// TIA Portal project "Lab_3" (V18)

(* hardware
DEVICE "S7-1500/ET200MP station_1"  S7-1500 station
   slot 0: "Rail_0"  Rack  6ES7 590-1***0-0AA0
   slot 1: "PLC_1"  CPU 1511-1 PN  6ES7 511-1AK00-0AB0  V1.0
      slot 3: "CPU display_1"  6ES7591-1XA00-0AA0
      slot 32768: "PROFINET interface_1"  X1
   slot 2: "CM 1542-5_1"  CM 1542-5  6GK7 542-5DX00-0XE0  V1.0
   slot 3: "DI 16x24VDC HF_1"  DI 16x24VDC HF  6ES7 521-1BH00-0AB0  V1.0
   slot 4: "DQ 16x24VDC/0.5A ST_1"  DQ 16x24VDC/0.5A ST  6ES7 522-1BH00-0AB0  V1.0
   slot 5: "AI 8xU/I/RTD/TC ST_1"  AI 8xU/I/RTD/TC ST  6ES7 531-7KF00-0AB0  V1.0
   slot 6: "AQ 4xU/I ST_1"  AQ 4xU/I ST  6ES7 532-5HD00-0AB0  V1.0
DEVICE "HMI_1"  KTP600 Basic color PN SIPLUS
   slot 0: "HMI_1"  KTP600 Basic color PN SIPLUS  6AG1 647-0AD11-2AX0  12.0.0.0
   slot 1: "HMI_RT_1"  KTP600 Basic color PN SIPLUS  6AG1 647-0AD11-2AX0  12.0.0.0
   slot 5: "HMI_1.IE_CP_1"  PROFINET Interface  12.0.0.0
      slot 1: "PROFINET Interface_1"  PROFINET Interface
         slot 1: "Port_1"  Port
*)

// ===== PLC "PLC_1"  CPU 1511-1 PN =====

VAR_GLOBAL   // PLC tag table "Default tag table"
   "Start_Pulse" AT %M0.0 : Bool;
   "En_Pulse" AT %M0.1 : Bool;
   "Low_Pulse_Active" AT %M0.2 : Bool;
   "High_Pulse_Enable" AT %M0.3 : Bool;
   "High_Pulse_Active" AT %M0.4 : Bool;
   "Low_Pulse_Enable" AT %M0.5 : Bool;
   "Pulse" AT %Q0.0 : Bool;
   "Start" AT %I0.0 : Bool;
   "Stop" AT %I0.1 : Bool;
   "Emergency" AT %I0.2 : Bool;
   "En_Bottle" AT %M2.0 : Bool;
   "R_Bottle" AT %M2.1 : Bool;
   "Finish_Bottle" AT %M2.2 : Bool;
   "Count_Bottle" AT %MW3 : Int;
   "R_Pulse" AT %M5.0 : Bool;
   "F_Pulse" AT %M5.1 : Bool;
   "Count_Pulse" AT %MW6 : Int;
   "En_PWM" AT %M8.0 : Bool;
   "Completo_PWM" AT %M8.1 : Bool;
   "T_PWM" AT %MD10 : Time;
   "E_Fill" AT %M14.0 : Bool;
   "Total_Fill" AT %M14.1 : Bool;
   "T_Fill" AT %MD15 : Time;
   "Valve" AT %M20.0 : Bool;
   "Bottles" AT %MW30 : Int;
   "Etapa" AT %M40.2 : Bool;
END_VAR

DATA_BLOCK "Generador_DB"   // DB2
{ S7_Optimized_Access := 'TRUE' }
VERSION : 0.1
// stored: InstanceOfName Generador
"Generador"
BEGIN
END_DATA_BLOCK

DATA_BLOCK "Contadores y Temporizadores_DB"   // DB3
{ S7_Optimized_Access := 'TRUE' }
VERSION : 0.1
// stored: InstanceOfName Contadores y Temporizadores
"Contadores y Temporizadores"
BEGIN
END_DATA_BLOCK

DATA_BLOCK "graph_DB"   // DB4
{ S7_Optimized_Access := 'TRUE' }
VERSION : 0.1
// stored: InstanceOfName graph
"graph"
BEGIN
END_DATA_BLOCK

FUNCTION_BLOCK "Generador"   // FB1, STL
{ S7_Optimized_Access := 'TRUE' }
VERSION : 0.1
   VAR
      IEC_Timer_0_Instance : TON_LTIME;
      DB1 : TON_LTIME;
   END_VAR
BEGIN

REGION Network 1
   // Habilitación
         A     "Start_Pulse";
         =     "En_Pulse";

   // Enable T1
         A     "En_Pulse";
         AN    "Low_Pulse_Active";
         =     "High_Pulse_Enable";

         CALL  #DB1
         ( IN := "High_Pulse_Enable",
           PT := LT#25000ns,
           Q  := "High_Pulse_Active",
           ET :=
         );



   // Enable T2
         A     "En_Pulse";
         A     "High_Pulse_Active";
         =     "Low_Pulse_Enable";

         CALL  #IEC_Timer_0_Instance
         ( IN := "Low_Pulse_Enable",
           PT := LT#25000ns,
           Q  := "Low_Pulse_Active",
           ET :=
         );


   // Salida
         A     "High_Pulse_Active";
         =     "Pulse";
END_REGION
END_FUNCTION_BLOCK

FUNCTION_BLOCK "Contadores y Temporizadores"   // FB3, SCL
{ S7_Optimized_Access := 'TRUE' }
VERSION : 0.1
   VAR RETAIN
      IEC_Counter_0_Instance : CTU_INT;
      IEC_Counter_0_Instance_1 : CTU_INT;
   END_VAR
   VAR
      IEC_Timer_0_Instance : TON_TIME;
      IEC_Timer_0_Instance_1 : TON_TIME;
   END_VAR
BEGIN
   #IEC_Counter_0_Instance(CU := "En_Bottle",
                           R := "R_Bottle",
                           PV := 32,   
                           Q => "Finish_Bottle",
                           CV => "Count_Bottle");

   #IEC_Counter_0_Instance_1(CU := "Pulse",
                             R := "R_Pulse",
                             PV := 500,
                             Q => "F_Pulse",
                             CV => "Count_Pulse");

   #IEC_Timer_0_Instance_1(IN:="E_Fill",
                           PT:=T#3s,
                           Q=>"Total_Fill",
                           ET=>"T_Fill");
   IF "Start" = 1 THEN
       // Statement section IF
       "Etapa" := TRUE;
       ;
   END_IF;

   IF "Stop" = 1 THEN
       // Statement section IF
       "Etapa" := FALSE;
   ELSE
       "Etapa" := TRUE;
       ;
   END_IF;

   IF "Emergency" = 1 THEN
       // Statement section IF
       "Etapa" := FALSE;
       "R_Bottle" := TRUE;
       "R_Pulse" := TRUE;
       "Valve" := FALSE;
       "En_PWM" := FALSE;
       "E_Fill" := FALSE;

       ;
   END_IF;
END_FUNCTION_BLOCK

FUNCTION_BLOCK "graph"   // FB4, GRAPH_PLUS
{ S7_Optimized_Access := 'TRUE' }
VERSION : 0.1
   VAR_INPUT
      OFF_SQ : Bool := false;   // Turn sequence off
      INIT_SQ : Bool := false;   // Set sequence to initial state
      ACK_EF : Bool := false;   // Acknowledge all errors and faults
      S_PREV : Bool := false;   // Output previous step in parameter S_NO
      S_NEXT : Bool := false;   // Indicate next step in parameter S_NO
      SW_AUTO : Bool := false;   // Automatic mode
      SW_TAP : Bool := false;   // Semiautomatic/switch with transition
      SW_TOP : Bool := false;   // Semiautomatic/ignore transition
      SW_MAN : Bool := false;   // Manual mode
      S_SEL : Int := 0;   // Select step to be output to S_NO
      S_ON : Bool := false;   // Activate step indicated in S_NO
      S_OFF : Bool := false;   // Disable step indicated in S_NO
      T_PUSH : Bool := false;   // Enable transition to switch in semi automatic mode
   END_VAR
   VAR_OUTPUT
      S_NO : Int := 0;   // Step number
      S_MORE : Bool := false;   // More steps are available and can be shown in S_NO
      S_ACTIVE : Bool := false;   // Step indicated in S_NO is active
      ERR_FLT : Bool := false;   // Interlock or supervision group error
      AUTO_ON : Bool := false;   // Automatic mode is active
      TAP_ON : Bool := false;   // Semiautomatic mode/step with transition enabled
      TOP_ON : Bool := false;   // Semiautomatic mode/ignore transition enabled
      MAN_ON : Bool := false;   // Manual mode is active
   END_VAR
   VAR
      HMI_INFO : Array[0..8] of UInt;
      IF_PAR : G7_IfParPlus_V2;
      RT_DATA : G7_RTDataPlus_V2;   // Internal data area
      Trans1 : G7_TransitionPlus_V2;   // Transition structure
      Trans3 : G7_TransitionPlus_V2;   // Transition structure
      Trans4 : G7_TransitionPlus_V2;   // Transition structure
      Trans5 : G7_TransitionPlus_V2;   // Transition structure
      Trans6 : G7_TransitionPlus_V2;   // Transition structure
      Trans7 : G7_TransitionPlus_V2;   // Transition structure
      Trans8 : G7_TransitionPlus_V2;   // Transition structure
      Trans9 : G7_TransitionPlus_V2;   // Transition structure
      Step1 : G7_StepPlus_V2;   // Step structure
      Step2 : G7_StepPlus_V2;   // Step structure
      Step3 : G7_StepPlus_V2;   // Step structure
      Step4 : G7_StepPlus_V2;   // Step structure
      Step5 : G7_StepPlus_V2;   // Step structure
      SINI : Array[0..1] of USInt;
      LSTT : Array[0..7] of USInt;
      ATAJ : Array[0..7] of USInt;
      ATAB : Array[0..7] of USInt;
      PSTT : Array[0..7] of USInt;
      NSTT : Array[0..7] of USInt;
      ASSJ : Array[0..4] of USInt;
      ASSB : Array[0..4] of USInt;
      PTTS : Array[0..4] of USInt;
      NTTS : Array[0..4] of USInt;
      SW_SQTS : Array[0..4] of USInt;
      SWITCH : Array[0..1] of USInt;
      TVX : Array[0..7] of USInt;
      TTX : Array[0..7] of USInt;
      TSX : Array[0..1] of USInt;
      S00X : Array[0..1] of USInt;
      SOFFX : Array[0..1] of USInt;
      SONX : Array[0..1] of USInt;
      SAX : Array[0..1] of USInt;
      SERRX : Array[0..5] of USInt;
      SMX : Array[0..5] of USInt;
      S0X : Array[0..5] of USInt;
      S1X : Array[0..5] of USInt;
      IL_ALARM_INST : Program_Alarm;
      SUP_ALARM_INST : Program_Alarm;
      STEP_TIME_ALARM_INST : Program_Alarm;
      IEC_TIMER_INST : IEC_TIMER;
      TRANSACTION_FLAG : Bool := false;
   END_VAR
   // LSTT[1] := 255;
   // SINI[0] := 2;
   // LSTT[0] := 255;
   // LSTT[3] := 255;
   // LSTT[5] := 1;
   // LSTT[6] := 255;
   // ATAJ[1] := 1;
   // ATAJ[2] := 2;
   // ATAJ[3] := 3;
   // ATAJ[4] := 4;
   // ATAJ[5] := 5;
   // ATAJ[6] := 6;
   // ATAJ[7] := 7;
   // ATAB[1] := 2;
   // ATAB[2] := 1;
   // ATAB[3] := 4;
   // ATAB[4] := 3;
   // ATAB[5] := 6;
   // ATAB[6] := 5;
   // ATAB[7] := 7;
   // NSTT[1] := 2;
   // PSTT[2] := 1;
   // PSTT[3] := 2;
   // PSTT[4] := 2;
   // PSTT[5] := 3;
   // PSTT[6] := 3;
   // PSTT[7] := 4;
   // PSTT[1] := 1;
   // NSTT[0] := 1;
   // NSTT[3] := 3;
   // NSTT[5] := 1;
   // NSTT[6] := 4;
   // ASSJ[1] := 1;
   // ASSJ[2] := 2;
   // ASSJ[3] := 3;
   // ASSJ[4] := 4;
   // ASSB[1] := 1;
   // ASSB[2] := 2;
   // ASSB[3] := 3;
   // ASSB[4] := 4;
   // PTTS[0] := 255;
   // PTTS[2] := 1;
   // PTTS[3] := 3;
   // PTTS[4] := 6;
   // NTTS[1] := 1;
   // NTTS[2] := 3;
   // NTTS[3] := 5;
   // NTTS[4] := 7;
   // SW_SQTS[2] := 1;
   // SW_SQTS[3] := 2;
   // SW_SQTS[4] := 3;
   // TVX[0] := 16#1;
   // TTX[0] := 16#1;
   // TSX[0] := 16#1;
   // S00X[0] := 16#1;
   // SOFFX[0] := 16#1;
   // SONX[0] := 16#1;
   // SAX[0] := 16#1;
   // SERRX[0] := 16#1;
   // SMX[0] := 16#1;
   // S0X[0] := 16#1;
   // S1X[0] := 16#1;
BEGIN
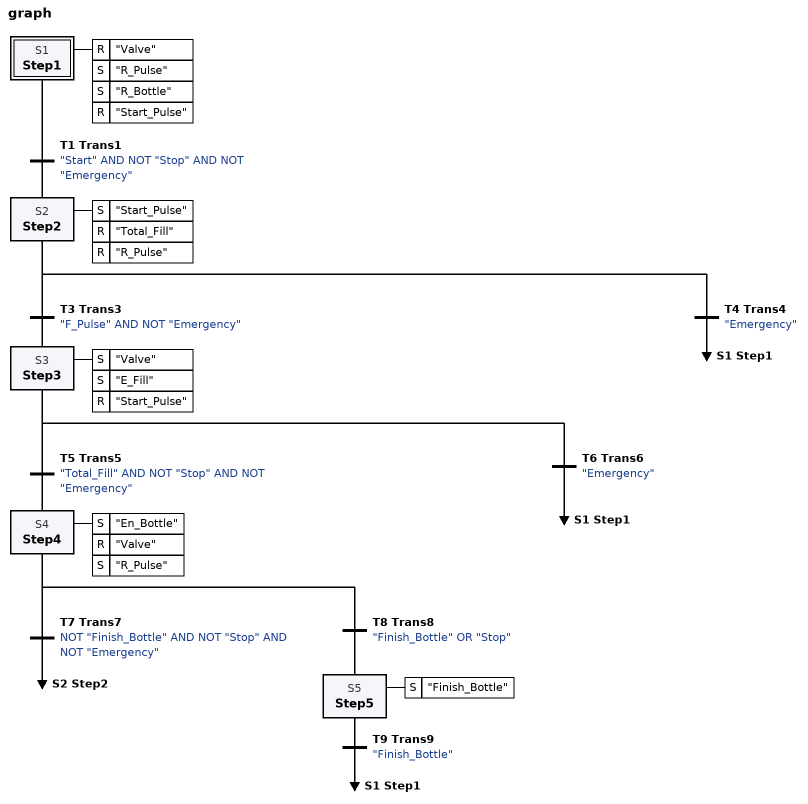
   // sequencer 1
   INITIAL_STEP Step1:   // S1, max time T#10S, warning time T#7S
              R    "Valve"
              S    "R_Pulse"
              S    "R_Bottle"
              R    "Start_Pulse"
   END_STEP
   TRANSITION Trans1 FROM Step1 TO Step2   // T1
      := "Start" AND NOT "Stop" AND NOT "Emergency";
   END_TRANSITION
   STEP Step2:   // S2, max time T#10S, warning time T#7S
              S    "Start_Pulse"
              R    "Total_Fill"
              R    "R_Pulse"
   END_STEP
   TRANSITION Trans3 FROM Step2 TO Step3   // T3
      := "F_Pulse" AND NOT "Emergency";
   END_TRANSITION
   TRANSITION Trans4 FROM Step2 TO Step1   // T4, jump
      := "Emergency";
   END_TRANSITION
   STEP Step3:   // S3, max time T#10S, warning time T#7S
              S    "Valve"
              S    "E_Fill"
              R    "Start_Pulse"
   END_STEP
   TRANSITION Trans5 FROM Step3 TO Step4   // T5
      := "Total_Fill" AND NOT "Stop" AND NOT "Emergency";
   END_TRANSITION
   TRANSITION Trans6 FROM Step3 TO Step1   // T6, jump
      := "Emergency";
   END_TRANSITION
   STEP Step4:   // S4, max time T#10S, warning time T#7S
              S    "En_Bottle"
              R    "Valve"
              S    "R_Pulse"
   END_STEP
   TRANSITION Trans7 FROM Step4 TO Step2   // T7, jump
      := NOT "Finish_Bottle" AND NOT "Stop" AND NOT "Emergency";
   END_TRANSITION
   TRANSITION Trans8 FROM Step4 TO Step5   // T8
      := "Finish_Bottle" OR "Stop";
   END_TRANSITION
   STEP Step5:   // S5, max time T#10S, warning time T#7S
              S    "Finish_Bottle"
   END_STEP
   TRANSITION Trans9 FROM Step5 TO Step1   // T9, jump
      := "Finish_Bottle";
   END_TRANSITION
END_FUNCTION_BLOCK

ORGANIZATION_BLOCK "Main"   // OB1, LAD, ProgramCycle
TITLE = "Main Program Sweep (Cycle)"
{ S7_Optimized_Access := 'TRUE' }
VERSION : 0.1
   VAR_INPUT
      Initial_Call : Bool;   // Initial call of this OB
      Remanence : Bool;   // =True, if remanent data are available
   END_VAR
BEGIN

REGION Network 1
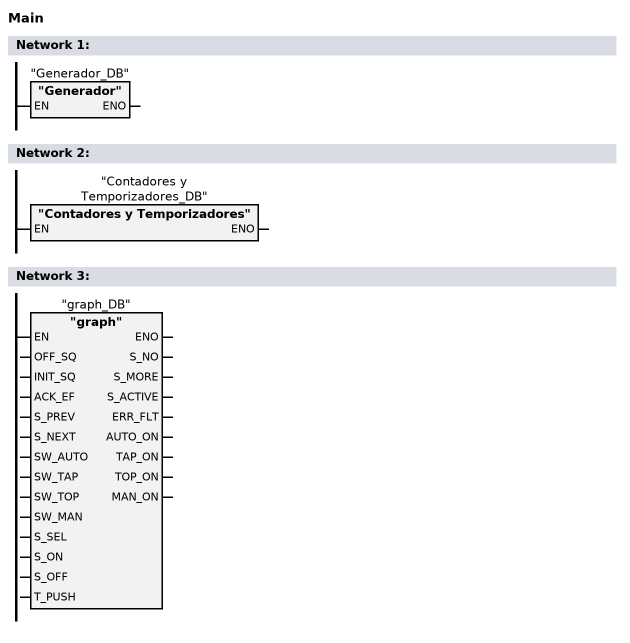
   RUNG wire#powerrail
      "Generador_DB"()
   END_RUNG
   // the same network as SCL:
   "Generador_DB"();   // "Generador"
END_REGION

REGION Network 2
   RUNG wire#powerrail
      "Contadores y Temporizadores_DB"()
   END_RUNG
   // the same network as SCL:
   "Contadores y Temporizadores_DB"();   // "Contadores y Temporizadores"
END_REGION

REGION Network 3
   RUNG wire#powerrail
      "graph_DB"(OFF_SQ :=, INIT_SQ :=, ACK_EF :=, S_PREV :=, S_NEXT :=, SW_AUTO :=, SW_TAP :=, SW_TOP :=, SW_MAN :=, S_SEL :=, S_ON :=, S_OFF :=, T_PUSH :=, S_NO =>, S_MORE =>, S_ACTIVE =>, ERR_FLT =>, AUTO_ON =>, TAP_ON =>, TOP_ON =>, MAN_ON =>)
   END_RUNG
   // the same network as SCL:
   "graph_DB"();   // "graph"
END_REGION
END_ORGANIZATION_BLOCK

(* ===== HMI "HMI_RT_1" =====
system functions are stored by id; their names below are inferred from use
connection "HMI_Connection_1": ETHERNET, SMART_S7_1500_OMS

HMI tags "Default tag table"
   "Tag_ScreenNumber" : UInt, internal
   "Start" : Bool = PLC Start AT %I0.0, 1 s
   "Stop" : Bool = PLC Stop AT %I0.1, 1 s
   "Emergency" : Bool = PLC Emergency AT %I0.2, 1 s

Template "Template_1" 320x240
   Button "Exit" at 266,202 size 52x37; TextOff 'Exit'; PictureOff "ExitRuntime_KTP600_Basic_color_PN"; PictureOn "ExitRuntime_KTP600_Basic_color_PN"
      on Release: StopRuntime(0)
   Button "Template_Button" at 213,202 size 52x37; TextOff 'Text'
   Button "Template_Button_1" at 160,202 size 52x37; TextOff 'Text'
   Button "Template_Button_2" at 107,202 size 52x37; TextOff 'Text'
   Button "Template_Button_3" at 54,202 size 52x37; TextOff 'Text'
   Button "Start screen" at 1,202 size 52x37; TextOff 'Start screen'; PictureOff "NavigateHome_KTP600_Basic_color_PN"; PictureOn "NavigateHome_KTP600_Basic_color_PN"
      on Release: ActivateScreen("Screen_1", 0)
   SymbolicIOField "Symbolic_IO_Field_Screen" at 69,7 size 164x24; TextOff '0'; TextOn '1'; TextList "TextList_ScreenNames"
      ProcessValue <- "Tag_ScreenNumber"
      on Change: ActivateScreenByNumber("Tag_ScreenNumber", 0)
   DateTimeField "HmiScreenItemData" at 235,19 size 85x19
   DateTimeField "HmiScreenItemData_1" at 235,0 size 85x19
   GraphicView "Logo" at 0,0 size 67x38; Picture "Logo of HMI_1"

screen "Screen_1" 320x240
   TextField "Text field_1" at 65,3 size 188x21; Text 'Sistema de Rectificado'
   Circle "Circle_1" at 4,70 size 32x32
      Appearance <- "Start"
   Circle "Circle_2" at 4,114 size 32x32
      Appearance <- "Stop"
   Circle "Circle_3" at 4,160 size 32x32
      Appearance <- "Emergency"
   IOField "I/O field_1" at 214,54 size 96x23
   IOField "I/O field_2" at 214,81 size 96x23
   IOField "I/O field_3" at 214,110 size 96x23
*)